Yaskawa INFORM job: DEMONSTRATOR_A6.JBI

/JOB
//NAME DEMONSTRATOR_A6
///FOLDERNAME DEMONSTRATOR
//POS
///NPOS 0,0,0,1,0,0
///USER 4
///TOOL 1
///POSTYPE USER
///RECTAN
///RCONF 1,0,0,0,0,0,0,0,0,0,0,0,0,0,0,0,0,0,0,0,0,0,0,0
P00100=-51.450,-41.710,12.601,0.0000,0.0000,0.0000
//ALIAS
///LVARS 0,2,26,0,0,0,0,0
LI000 Point
LI001 Direction
LD000 HALBKREIS
LD001 X_right
LD002 Y_upper
LD003 MX
LD004 MY
LD005 RADIUS
LD006 Y_lower
LD007 X_offset
LD008 X
LD009 X_left
LD010 Z_left
LD011 Z_right
LD012 USERFRAME
LD013 Z_offset
LD014 Width
LD015 Beads_inner
LD016 Z
LD017 X_mirror
LD018 V_weld
LD019 KENNLINIE
LD020 V_weld_offset
LD021 X_left_inner
LD022 X_right_inner
LD023 Beads_outer
LD024 Spurbreite
LD025 Uebermass
//ARGINFO
///ARGTYPE D,D,D,D,D,D,D,D
///COMMENT
X left
X right
X Offset
Height_left
Height_right
USERFRAME
V_WELD
Kennlinie
//INST
///DATE 2023/01/24 14:22
///ATTR SC,RW
///GROUP1 RB1
///LVARS 1,3,27,0,0,0,0,0
NOP
TCPON TL#(0)
CALL JOB:SET_TCPON ARGF0
'################################
'Einlesen der Argumente
GETARG X_left IARG#(1)
GETARG X_right IARG#(2)
GETARG X_offset IARG#(3)
GETARG Z_left IARG#(4)
GETARG Z_right IARG#(5)
GETARG USERFRAME IARG#(6)
GETARG V_weld IARG#(7)
GETARG KENNLINIE IARG#(8)
'################################
SET V_weld_offset  EXPRESS V_weld * 2
'################################
SET Z Z_left
SET Point 0
SET Direction 1
SET Spurbreite 9000
SET Uebermass 4000
'################################
'Berechnen der fertigbaren Breite
' Width = vielfaches von x_Offset
' Gerade Anzahl von Raupen
SET Beads_outer  EXPRESS ( X_right - X_left ) / ( X_offset )
CALL JOB:GET_EVEN_NUMBER ARGFBeads_outer ARGF"DOWN"
GETS Beads_outer $RV
ADD Beads_outer 1
SET Width  EXPRESS X_offset * Beads_outer
'################################
'################################
'Berechnen der inneren Grenezen
SET X_left_inner  EXPRESS Width * -0.5
WHILEEXP X_left_inner<-51070
	 ADD X_left_inner X_offset
ENDWHILE
SET X_right_inner X_left_inner
WHILEEXP X_right_inner<-22500
	 ADD X_right_inner X_offset
ENDWHILE
SUB X_right_inner X_offset
'Berechnung der Anzahl der
'Punkte in der Teilflaeche
'Fehlermeldung if P>98 -->
'98 globale Punktvariablen
SET Beads_inner  EXPRESS ( X_right_inner - X_left_inner ) / ( X_offset )
SET Point  EXPRESS Beads_inner * 2
IFTHENEXP Point>98
	 SET B000  EXPRESS 400
	 MSG "STRING"
ENDIF
'################################
'Kontrolle
SET D030 Width
SET D031 X_left_inner
SET D032 X_right_inner
SET D033 Beads_outer
SET D034 Beads_inner
SET D035  EXPRESS X_right_inner - X_left_inner
SET D036  EXPRESS D035 / D034
'###############################
SET Z_offset  EXPRESS ( Z_right - Z_left ) / ( Beads_inner )
SET Point 0
SET X X_left_inner
WHILEEXP X<=X_right_inner
	 SET MX 0
	 SET MY 640000
	 SET RADIUS 600000
	 SET HALBKREIS -1
	 CALL JOB:GET_KREISKOORDINATEN ARGFX ARGFMX ARGFMY ARGFRADIUS ARGFHALBKREIS
	 GETS Y_upper $RV
	 SET Y_upper  EXPRESS Y_upper - 0.5 * Spurbreite + Uebermass
	'untere Kontur (Kreis)
	 SET MX 0
	 SET MY -640000
	 SET RADIUS 600000
	 SET HALBKREIS 1
	 CALL JOB:GET_KREISKOORDINATEN ARGFX ARGFMX ARGFMY ARGFRADIUS ARGFHALBKREIS
	 GETS Y_lower $RV
	 SET Y_lower  EXPRESS Y_lower + 0.5 * Spurbreite - Uebermass
	 SET X_mirror  EXPRESS X * -1
	'Punkte schreiben
	 IFTHENEXP Direction=1
		 CALL JOB:PUNKTE_ERZEUGEN_UF ARGFUSERFRAME ARGFX_mirror ARGFY_lower ARGFZ
		 SET P[Point] P100
		 ADD Point 1
		 CALL JOB:PUNKTE_ERZEUGEN_UF ARGFUSERFRAME ARGFX_mirror ARGFY_upper ARGFZ
		 SET P[Point] P100
		 ADD Point 1
		 MUL Direction -1
	 ELSEIFEXP Direction=-1
		 CALL JOB:PUNKTE_ERZEUGEN_UF ARGFUSERFRAME ARGFX_mirror ARGFY_upper ARGFZ
		 SET P[Point] P100
		 ADD Point 1
		 CALL JOB:PUNKTE_ERZEUGEN_UF ARGFUSERFRAME ARGFX_mirror ARGFY_lower ARGFZ
		 SET P[Point] P100
		 ADD Point 1
		 MUL Direction -1
	 ENDIF
	 SET I001 Point
	 ADD Z Z_offset
	 ADD X X_offset
ENDWHILE
'########################
'##########Welding#######
CALL JOB:DEMONSTRATOR_WELD_MEAND ARGFPoint ARGFV_weld ARGFKENNLINIE ARGF62
END
